{attribute addProperty BoxType "EL3632-0000-0016"}
{attribute addProperty Id "Ch1_ValueAT %I*INT162"}
{attribute addProperty CRC "935361667"}
{attribute addProperty SizeInBites "16"}
{attribute addProperty SizeInBytes "2"}
TYPE Ch1_Sample_37C07C83 :
STRUCT
	{attribute addProperty Name "Ch1_Value"}
	Ch1_Value AT %I* : INT;
END_STRUCT
END_TYPE

(* stored: Version 1.2.0.0, ProductVersion 3.1.4024.9
   DUT Ch1_Sample_37C07C83: Id {d4d46d28-9872-4d3b-9f4e-d8cf5a8c3853} *)
